Omron CX-Programmer project NewProject (CX-Programmer 9.51)

# PLC NewPLC1: CP1L L
; MyFirstProject

## Global symbols (name address type ; comment)
1 CHANNEL  ; comment
5 CHANNEL  ; comment
C0001 BOOL  ; #5

## Program NewProgram1 (cyclic task 0)
Local symbols
I 0.00 BOOL  ; Input1
Q 100.01 BOOL  ; Output2
button1 0.00 BOOL
zz UINT

### Section Section1

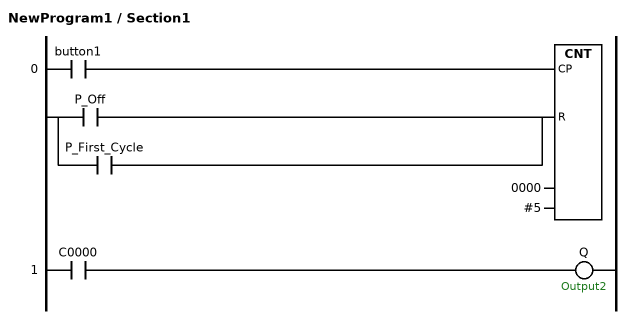
; rung 0
LD button1
LD P_Off
OR P_First_Cycle
CNT 0000 #5
; rung 1
LD C0000
OUT Q  ; Output2

### Section END
; rung 0
END(001)